FUNCTION_BLOCK bfb_controller_um
  (* Standard: 61499-2 *)
  (* Version 0.1, 2018-00-09, palme, DESKTOP-TGOEKBD *)
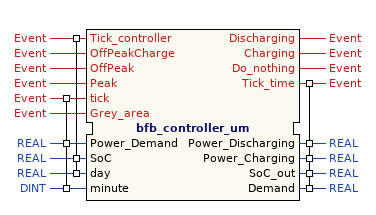
  EVENT_INPUT
    Tick_controller WITH SoC, day;
    OffPeakCharge;
    OffPeak;
    Peak;
    tick WITH Power_Demand, minute;
    Grey_area;
  END_EVENT
  EVENT_OUTPUT
    Discharging;
    Charging;
    Do_nothing;
    Tick_time WITH Power_Discharging, Power_Charging, SoC_out, Demand;
  END_EVENT
  VAR_INPUT
    Power_Demand : REAL;
    SoC : REAL;
    day : REAL;
    minute : DINT;
  END_VAR
  VAR_OUTPUT
    Power_Discharging : REAL;
    Power_Charging : REAL;
    SoC_out : REAL;
    Demand : REAL;
  END_VAR
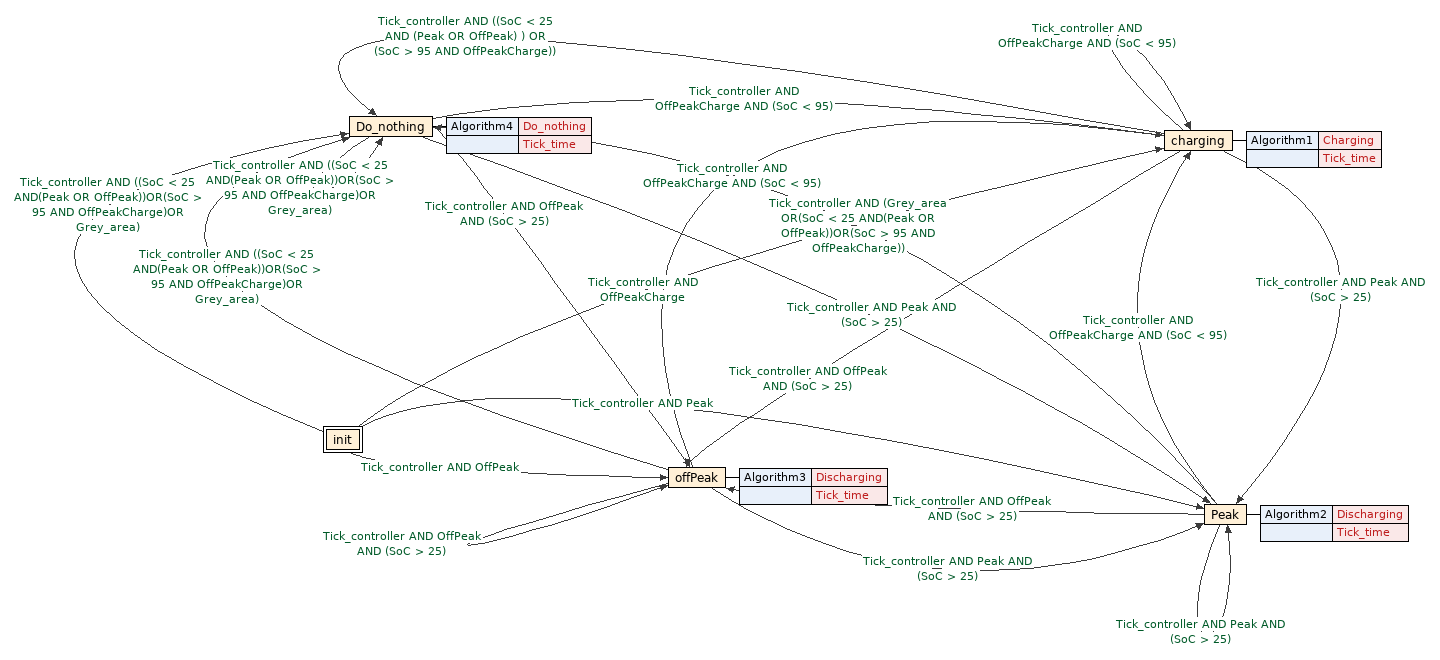
  EC_STATES
    init;
    Do_nothing : Algorithm4 -> Do_nothing, -> Tick_time;
    charging : Algorithm1 -> Charging, -> Tick_time;
    Peak : Algorithm2 -> Discharging, -> Tick_time;
    offPeak : Algorithm3 -> Discharging, -> Tick_time;
  END_STATES
  EC_TRANSITIONS
    Do_nothing TO charging := Tick_controller AND OffPeakCharge AND (SoC < 95);
    Do_nothing TO Peak := Tick_controller AND Peak AND (SoC > 25);
    Do_nothing TO offPeak := Tick_controller AND OffPeak AND (SoC > 25);
    Do_nothing TO Do_nothing := Tick_controller AND ((SoC < 25 AND(Peak OR OffPeak))OR(SoC > 95 AND OffPeakCharge)OR Grey_area);
    charging TO Do_nothing := Tick_controller AND ((SoC < 25 AND (Peak OR OffPeak) ) OR (SoC > 95 AND OffPeakCharge));
    charging TO Peak := Tick_controller AND Peak AND (SoC > 25);
    charging TO offPeak := Tick_controller AND OffPeak AND (SoC > 25);
    charging TO charging := Tick_controller AND OffPeakCharge AND (SoC < 95);
    Peak TO offPeak := Tick_controller AND OffPeak AND (SoC > 25);
    Peak TO charging := Tick_controller AND OffPeakCharge AND (SoC < 95);
    Peak TO Do_nothing := Tick_controller AND (Grey_area OR(SoC < 25 AND(Peak OR OffPeak))OR(SoC > 95 AND OffPeakCharge));
    Peak TO Peak := Tick_controller AND Peak AND (SoC > 25);
    offPeak TO Peak := Tick_controller AND Peak AND (SoC > 25);
    offPeak TO charging := Tick_controller AND OffPeakCharge AND (SoC < 95);
    offPeak TO Do_nothing := Tick_controller AND ((SoC < 25 AND(Peak OR OffPeak))OR(SoC > 95 AND OffPeakCharge)OR Grey_area);
    offPeak TO offPeak := Tick_controller AND OffPeak AND (SoC > 25);
    init TO Do_nothing := Tick_controller AND ((SoC < 25 AND(Peak OR OffPeak))OR(SoC > 95 AND OffPeakCharge)OR Grey_area);
    init TO offPeak := Tick_controller AND OffPeak;
    init TO charging := Tick_controller AND OffPeakCharge;
    init TO Peak := Tick_controller AND Peak;
  END_TRANSITIONS
  ALGORITHM Algorithm1 IN C:
me->Power_Charging = 200;
printf(" Controler Charging state  \r\n");
//me->SoC_out = me->SoC;
//printf("Power Charging: %f", me->Power_Charging);
REAL Day = me->day;
DINT Minute = me->minute;

REAL Demand = me->Power_Demand;
me->Demand = Demand;
printf("Minute = %d Demand = %f",Minute, Demand);

if (Minute == 0 && Day == 0){
me->SoC = 90;
}
else{
me->SoC_out = me->SoC;
}
  END_ALGORITHM
  ALGORITHM Algorithm2 IN C:
REAL Power_required = me->Power_Demand;
REAL max_ESS_discharge = 150;
REAL Day = me->day;
DINT Minute = me->minute;
REAL Demand = me->Power_Demand;
me->Demand = Demand;

printf("Minute = %d Demand = %f",Minute, Demand);
if (max_ESS_discharge >  Power_required){
me->Power_Discharging = Power_required;
}
else {
me->Power_Discharging = max_ESS_discharge;
}

if (Minute == 0 && Day == 0){
me->SoC = 90;
}
else{
me->SoC_out = me->SoC;
}
//me->SoC_out = me->SoC;
printf(" Disharging.... state..Controller \r\n ");
  END_ALGORITHM
  ALGORITHM Algorithm3 IN C:
REAL Power_required = me->Power_Demand;
REAL Peak = 130;
REAL max_ESS_discharge = 150;
REAL Day = me->day;
DINT Minute = me->minute;

printf("Minute1 = %d Demand1 = %f \r\n",Minute, Power_required);

if (Peak < Power_required){
	if (max_ESS_discharge > Power_required-Peak){
	me->Power_Discharging = Power_required - Peak;
	}
	else{
	me->Power_Discharging = max_ESS_discharge;
	}
}
else{
me->Power_Discharging = 0;
}
me->Demand = Power_required;
if (Minute == 0 && Day == 0){
me->SoC = 90;
}
else{
me->SoC_out = me->SoC;
}

//me->SoC_out = me->SoC;
printf(" Discharging.... state, OFFpeak controller \r\n ");
  END_ALGORITHM
  ALGORITHM Algorithm4 IN C:
REAL Day = me->day;
DINT Minute = me->minute;
printf("Do Nothing, controller \r\n");
REAL Demand = me->Power_Demand;
me->Demand = Demand;
printf("Minute = %d Demand = %f",Minute, Demand);
if (Minute == 0 && Day == 0){
//me->SoC = 0;
me->SoC_out = 90;
}
else{
me->SoC_out = me->SoC;
}
  END_ALGORITHM
END_FUNCTION_BLOCK
